// TIA Portal project "Project7" (V19)

(* hardware
DEVICE "S7-1200 station_1"  S7-1200 Station
   slot 0: "Rack_0"  S7-1200 Rack  Rack  V1.0
   slot 1: "PLC_1"  CPU 1214C DC/DC/DC  6ES7 214-1AG40-0XB0  V4.5
   slot 3: "CB 1241 (RS485)"  CB 1241 (RS485)  6ES7 241-1CH30-1XB0  V1.0
*)

// ===== PLC "PLC_1"  CPU 1214C DC/DC/DC =====

VAR_GLOBAL   // PLC tag table "Default tag table"
   "Clock_Byte" AT %MB0 : Byte;
   "Clock_10Hz" AT %M0.0 : Bool;
   "Clock_5Hz" AT %M0.1 : Bool;
   "Clock_2.5Hz" AT %M0.2 : Bool;
   "Clock_2Hz" AT %M0.3 : Bool;
   "Clock_1.25Hz" AT %M0.4 : Bool;
   "Clock_1Hz" AT %M0.5 : Bool;
   "Clock_0.625Hz" AT %M0.6 : Bool;
   "Clock_0.5Hz" AT %M0.7 : Bool;
   "System_Byte" AT %MB1 : Byte;
   "FirstScan" AT %M1.0 : Bool;
   "DiagStatusUpdate" AT %M1.1 : Bool;
   "AlwaysTRUE" AT %M1.2 : Bool;
   "AlwaysFALSE" AT %M1.3 : Bool;
END_VAR

DATA_BLOCK "Block_1_DB"   // DB1
{ S7_Optimized_Access := 'TRUE' }
VERSION : 0.1
// stored: InstanceOfName Block_1
"Block_1"
BEGIN
END_DATA_BLOCK

DATA_BLOCK "Status"   // DB3
{ S7_Optimized_Access := 'TRUE' }
VERSION : 0.1
   VAR
      Done : Bool;
      Err : Word;
      Move : Word;
      Err2 : Word;
      Move2 : Word;
   END_VAR
BEGIN
END_DATA_BLOCK

DATA_BLOCK "Datos"   // DB5
{ S7_Optimized_Access := 'FALSE' }
VERSION : 0.1
   VAR
      data : Array[0..5] of Bool;
   END_VAR
BEGIN
END_DATA_BLOCK

FUNCTION_BLOCK "Block_1"   // FB1, LAD
{ S7_Optimized_Access := 'TRUE' }
VERSION : 0.1
BEGIN

REGION Network 1
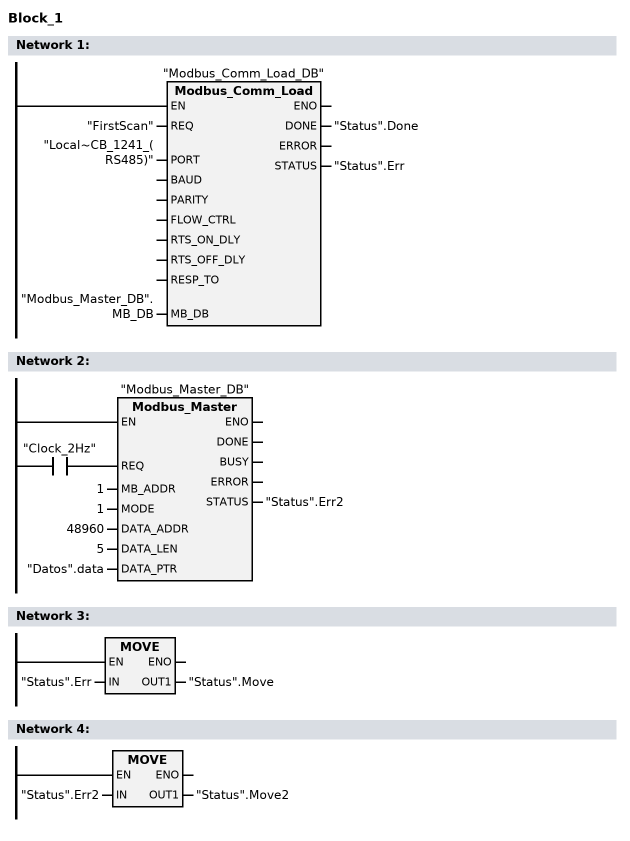
   "Modbus_Comm_Load_DB"(REQ := "FirstScan",   // Modbus_Comm_Load
                         PORT := "Local~CB_1241_(RS485)",
                         MB_DB := "Modbus_Master_DB".MB_DB,
                         DONE => "Status".Done,
                         STATUS => "Status".Err);
END_REGION

REGION Network 2
   "Modbus_Master_DB"(REQ := "Clock_2Hz",   // Modbus_Master
                      MB_ADDR := 1,
                      MODE := 1,
                      DATA_ADDR := 48960,
                      DATA_LEN := 5,
                      DATA_PTR := "Datos".data,
                      STATUS => "Status".Err2);
END_REGION

REGION Network 3
   RUNG wire#powerrail
      Move(in := "Status".Err, out1 => "Status".Move)
   END_RUNG
   // the same network as SCL:
   "Status".Move := "Status".Err;
END_REGION

REGION Network 4
   RUNG wire#powerrail
      Move(in := "Status".Err2, out1 => "Status".Move2)
   END_RUNG
   // the same network as SCL:
   "Status".Move2 := "Status".Err2;
END_REGION
END_FUNCTION_BLOCK

ORGANIZATION_BLOCK "Main"   // OB1, LAD, ProgramCycle
TITLE = "Main Program Sweep (Cycle)"
{ S7_Optimized_Access := 'TRUE' }
VERSION : 0.1
   VAR_INPUT
      Initial_Call : Bool;   // Initial call of this OB
      Remanence : Bool;   // =True, if remanent data are available
   END_VAR
BEGIN

REGION Network 1
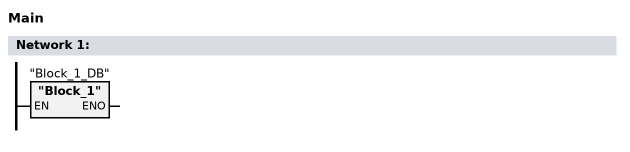
   RUNG wire#powerrail
      "Block_1_DB"()
   END_RUNG
   // the same network as SCL:
   "Block_1_DB"();   // "Block_1"
END_REGION
END_ORGANIZATION_BLOCK